FUNCTION_BLOCK pickup (* Basic Function Block Type *)
  (* Standard: 61499-2 *)
  (* Version 0.0, 10/19/2017, chivdan, nxtControl GmbH, Template *)
  PACKAGE Main;
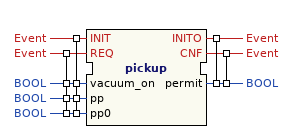
  EVENT_INPUT
    INIT WITH vacuum_on, pp, pp0; (* Initialization Request *)
    REQ WITH vacuum_on, pp, pp0; (* Normal Execution Request *)
  END_EVENT
  EVENT_OUTPUT
    INITO WITH permit; (* Initialization Confirm *)
    CNF WITH permit; (* Execution Confirmation *)
  END_EVENT
  VAR_INPUT
    vacuum_on : BOOL; (* Input event qualifier *)
    pp : BOOL;
    pp0 : BOOL;
  END_VAR
  VAR_OUTPUT
    permit : BOOL; (* Output event qualifier *)
  END_VAR
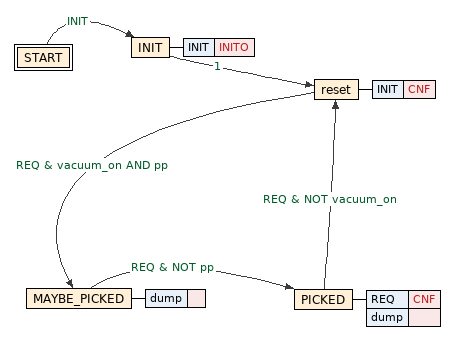
  EC_STATES
    START; (* Initial State *)
    INIT : INIT -> INITO; (* Initialization *)
    MAYBE_PICKED : dump; (* Normal execution *)
    PICKED : REQ -> CNF, dump;
    reset : INIT -> CNF;
  END_STATES
  EC_TRANSITIONS
    START TO INIT := INIT;
    reset TO MAYBE_PICKED := REQ & vacuum_on AND pp;
    MAYBE_PICKED TO PICKED := REQ & NOT pp;
    PICKED TO reset := REQ & NOT vacuum_on;
    INIT TO reset := 1;
  END_TRANSITIONS
  ALGORITHM INIT IN ST: (* Initialization algorithm *)
permit := TRUE;
  END_ALGORITHM
  ALGORITHM REQ IN ST: (* Normally executed algorithm *)
permit := FALSE;
  END_ALGORITHM
  ALGORITHM dump IN ST:
;
REQ:=FALSE;
  END_ALGORITHM
END_FUNCTION_BLOCK
